(* Logix 5000 project; controller WWTP_SOLIDS_CLX vendor 1 type 14 code 54 rev 17.2; software revision 17.00; part 9 of 16 *)
(* tags used below, declared in another part *)
   Inp_RunFdbk : BOOL;   // Input Signal: RUN feedback from motor
   Inp_PermOK : BOOL;   // 1=Permissives OK, motor can start
   Inp_NBPermOK : BOOL;   // 1=Non-Bypassable Permissives OK, motor can start
   Inp_IntlkOK : BOOL;   // 1=Interlocks OK, motor can start/run
   Inp_NBIntlkOK : BOOL;   // 1=Non-Bypassable Interlocks OK, motor can start/run
   Inp_IOFault : BOOL;   // Input Communication Status 0=OK, 1=fail
   Inp_Sim : BOOL;   // 1=Simulate working motor; 0=Start/Stop/ Monitor actual motor
   Inp_Hand : BOOL;   // 1=Select Hand (hardwired) Control Strategy
   Inp_Ovrd : BOOL;   // 1=Select Override control strategy
   Inp_OvrdState : BOOL;   // 1=Override to RUN, 0=Override to STOP
   Inp_Reset : BOOL;   // 1=Reset all fault conditions and latched Alarms
   Cfg_HasRunFdbk : BOOL;   // 1=Motor provides a run feedback signal
   Cfg_UseRunFdbk : BOOL;   // 1=Motor run feedback should be used for failure checking
   Cfg_PCmdClear : BOOL;   // 1=Clear Program Commands on receipt 0=Leave Set
   Cfg_OvrdPermIntlk : BOOL;   // 1=Override ignores Bypassable Perm/ Intlk; 0=always use Perm/Intlk
   Cfg_HasFailToStartAlm : BOOL;   // 1=Fail to Start Alarm exists and will be checked
   Cfg_HasFailToStopAlm : BOOL;   // 1=Fail to Stop Alarm exists and will be checked
   Cfg_HasIntlkTripAlm : BOOL;   // 1=Interlock Trip Alarm exists and will be checked
   Cfg_HasIOFaultAlm : BOOL;   // 1=I/O Fault Alarm exists and will be checked
   Cfg_FailToStartResetReqd : BOOL;   // 1=Reset required to clear Fail to Start Alarm
   Cfg_FailToStopResetReqd : BOOL;   // 1=Reset required to clear Fail to Stop Alarm
   Cfg_IntlkTripResetReqd : BOOL;   // 1=Reset required to clear Interlock Trip Alarm
   Cfg_IOFaultResetReqd : BOOL;   // 1=Reset required to clear I/O Fault Alarm
   Cfg_FailToStartAckReqd : BOOL;   // 1=Acknowledge required for Fail to Start Alarm
   Cfg_FailToStopAckReqd : BOOL;   // 1=Acknowledge required for Fail to Stop Alarm
   Cfg_IntlkTripAckReqd : BOOL;   // 1=Acknowledge required for Interlock Trip Alarm
   Cfg_IOFaultAckReqd : BOOL;   // 1=Acknowledge required for I/O Fault Alarm
   Cfg_FailToStartSeverity : SINT;   // Fail To Start Alarm Severity 1=info 2=warn 3=excep 4=fault
   Cfg_FailToStopSeverity : SINT;   // Fail To Stop Alarm Severity 1=info 2=warn 3=excep 4=fault
   Cfg_IntlkTripSeverity : SINT;   // Interlock Trip Alarm Severity 1=info 2=warn 3=excep 4=fault
   Cfg_IOFaultSeverity : SINT;   // I/O Fault Alarm Severity 1=info 2=warn 3=excep 4=fault
   Cfg_SimFdbkT : DINT;   // Delay to echo back of Running/Stopped status when in Simulation (sec)
   Cfg_FailToStartT : DINT;   // Time after Start to get Run Feedback before Fault (sec)
   Cfg_FailToStopT : DINT;   // Time after Stop to drop Run Feedback before Fault (sec)
   PSet_Owner : DINT;   // Program Owner Request ID (non-zero) or Release (zero)
   PCmd_Start : BOOL;   // Program Command to Start Motor
   PCmd_Stop : BOOL;   // Program Command to Stop Motor
   PCmd_Acq : BOOL;   // Program Command to Acquire ownership (Oper/OOS to Prog)
   PCmd_Rel : BOOL;   // Program Command to Release ownership (Prog to OOS)
   PCmd_Lock : BOOL;   // Program Command to Lock Mode in Prog
   PCmd_Unlock : BOOL;   // Program Command to Unlock Mode
   PCmd_Reset : BOOL;   // Program Command to Reset all Alarms requiring Reset
   PCmd_FailToStartAck : BOOL;   // Program Command to Acknowledge Fail to Start Alarm
   PCmd_FailToStartInhibit : BOOL;   // Program Command to Inhibit Fail to Start Alarm
   PCmd_FailToStartUninhibit : BOOL;   // Program Command to Uninhibit Fail to Start Alarm
   PCmd_FailToStopAck : BOOL;   // Program Command to Acknowledge Fail to Stop Alarm
   PCmd_FailToStopInhibit : BOOL;   // Program Command to Inhibit Fail to Stop Alarm
   PCmd_FailToStopUninhibit : BOOL;   // Program Command to Uninhibit Fail to Stop Alarm
   PCmd_IntlkTripAck : BOOL;   // Program Command to Acknowledge Interlock Trip Alarm
   PCmd_IntlkTripInhibit : BOOL;   // Program Command to Inhibit Interlock Trip Alarm
   PCmd_IntlkTripUninhibit : BOOL;   // Program Command to Uninhibit Interlock Trip Alarm
   PCmd_IOFaultAck : BOOL;   // Program Command to Acknowledge I/O Fault Alarm
   PCmd_IOFaultInhibit : BOOL;   // Program Command to Inhibit I/O Fault Alarm
   PCmd_IOFaultUninhibit : BOOL;   // Program Command to Uninhibit I/O Fault Alarm
   OCmd_Start : BOOL;   // Operator Command to Start Motor
   OCmd_Stop : BOOL;   // Operator Command to Stop Motor
   OCmd_Bypass : BOOL;   // Operator Command to Bypass all Bypassable Interlocks and Permissives
   OCmd_Check : BOOL;   // Operator Command to Check (not bypass) all Interlocks and Permissives
   MCmd_Disable : BOOL;   // Maintenance Command to Disable Motor
   MCmd_Enable : BOOL;   // Maintenance Command to Enable (allow to run) Motor
   OCmd_Reset : BOOL;   // Operator Command to Reset all Alarms requiring Reset
   Out_Run : BOOL;   // 1=Run Motor, 0=Stop Motor
   Out_Start : BOOL;   // 1=Start Motor, 0=Motor left in current state
   Out_Stop : BOOL;   // 1=Stop Motor, 0=Motor left in current state
   Val_Owner : DINT;   // Current Object Owner ID (0=not owned)
   Val_Notify : SINT;   // Current Alarm Level and Acknowledgement (enumeration)
   Sts_Disabled : BOOL;   // 1=Motor is Disabled
   Sts_Err : BOOL;   // 1=Error in Config: see detail bits for reason
   Err_Timer : BOOL;   // 1=Error in Config: Start/Stop Check timer preset (use 0 to 2147483)
   Err_Sim : BOOL;   // 1=Error in Config: Simulation timer preset (use 0 to 2147483)
   Err_Alarm : BOOL;   // 1=Error in Config: Invalid Alarm Severity
   Sts_Hand : BOOL;   // 1=Mode is Hand (supersedes Maint, Ovrd, Prog, Oper)
   Sts_Maint : BOOL;   // 1=Mode is Maintenance (supersedes Ovrd, Prog, Oper)
   Sts_Ovrd : BOOL;   // 1=Mode is Override (supersedes Prog, Oper)
   Sts_Prog : BOOL;   // 1=Mode is Program (auto)
   Sts_Oper : BOOL;   // 1=Mode is Operator (manual)
   Sts_ProgOperLock : BOOL;   // 1=Program or Operator has requested Mode Lock
   Sts_FailToStart : BOOL;   // 1=Motor Failed to Start (one-shot)
   Alm_FailToStart : BOOL;   // 1=Motor Fail to Start Alarm
   Ack_FailToStart : BOOL;   // 1=Fail to Start Alarm has been acknowledged
   Sts_FailToStartDisabled : BOOL;   // 1=Fail to Start Alarm has been disabled (will not be sent)
   Sts_FailToStartInhibited : BOOL;   // 1=Fail to Start Alarm has been inhibited by logic
   Sts_FailToStartSuppressed : BOOL;   // 1=Fail to Start Alarm has been suppressed (logged only)
   Sts_FailToStop : BOOL;   // 1=Motor Failed to Stop
   Alm_FailToStop : BOOL;   // 1=Motor Fail to Stop Alarm
   Ack_FailToStop : BOOL;   // 1=Fail to Stop Alarm has been acknowledged
   Sts_FailToStopDisabled : BOOL;   // 1=Fail to Stop Alarm has been disabled (will not be sent)
   Sts_FailToStopInhibited : BOOL;   // 1=Fail to Stop Alarm has been inhibited by logic
   Sts_FailToStopSuppressed : BOOL;   // 1=Fail to Stop Alarm has been suppressed (logged only)
   Sts_IntlkTrip : BOOL;   // 1=Motor stopped by an Interlock NOT OK (one-shot)
   Sts_IOFault : BOOL;   // I/O Comm Fault Status (0=OK, 1=Bad)
   Rdy_Reset : BOOL;   // 1=Ready to receive OCmd_Reset (enables HMI button)
   Mode : P_Mode;   // Motor Mode Selection
   IOFault : P_Alarm;   // I/O Fault Alarm
   IntlkTrip : P_Alarm;   // Interlock Trip Alarm
   FailToStop : P_Alarm;   // Motor Failed to Stop Alarm
   FailToStart : P_Alarm;   // Motor Failed to Start Alarm
   Wrk_Run : BOOL;   // 1=Motor should be "running", 0=should be "stopped"
   Wrk_SimRunT : TIMER;   // Simulation Delay until Running
   Wrk_StopT : TIMER;   // Stop Check Timer
   Wrk_StartT : TIMER;   // Start Check Timer
   Wrk_Fault : BOOL;   // 1=a Motor Fault has been detected
   Wrk_SimStopT : TIMER;   // Simulation Delay until Stopped
   Wrk_RunFdbk : BOOL;   // Run Feedback based on mode, simulation, etc. 1=running
   Wrk_IntlkTrip : BOOL;   // 1=Interlock Not OK Tripped Running Motor
   Wrk_Bypass : BOOL;   // Internal Bypassable Permissives and Interlocks are Bypassed flag
   Wrk_Disabled : BOOL;   // Internal Motor is Disabled
(* P_Motor, continued *)

ROUTINE Logic   (* ladder *)
// Normal Scan: control / monitor single speed motor
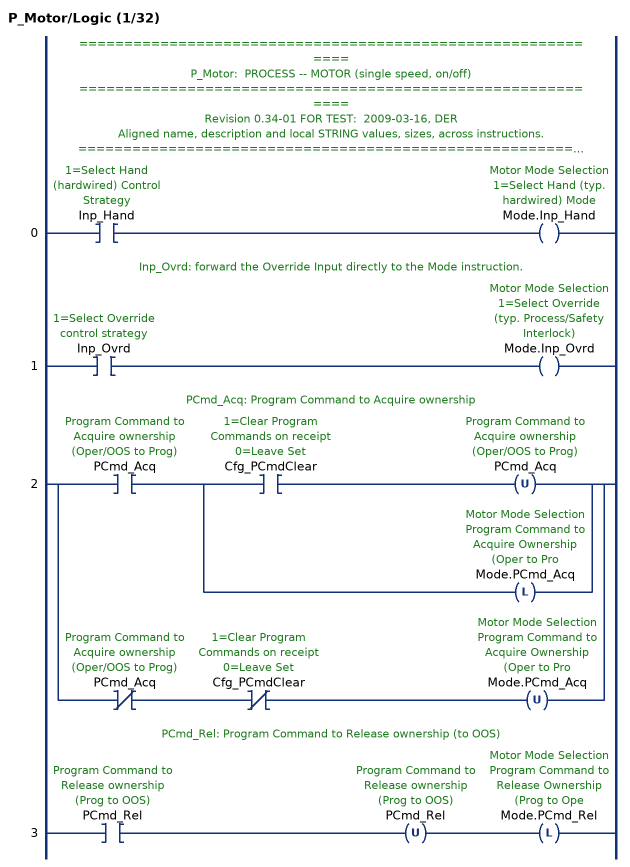
   // ============================================================
   // P_Motor:  PROCESS -- MOTOR (single speed, on/off)
   // ============================================================
   // Revision 0.34-01 FOR TEST:  2009-03-16, DER
   // Aligned name, description and local STRING values, sizes, across instructions.
   // ============================================================
   // This Instruction controls and monitors a single-speed motor
   // (FVNR, soft-start, etc.) and provides:
   // *  Monitoring of run feedback, display of actual motor status
   // *  Detection of Failure to Start, Failure to Stop
   // *  Monitoring of a Permissive condition to allow starting
   // * Monitoring of an Interlock condition to stop / prevent starting
   // * Simulation, providing feedback of a working motor while disabling outputs
   // * Monitoring of I/O communication faults
   // * Alarms for Fail to Start, Fail to Stop, Interlock Trip, I/O Fault
   // * Operation in Hand, Maintenance, Override, Program and Operator Modes
   // * "Available" status for use by automation logic to know whether motor
   // can be controlled by other objects.
   // ============================================================
   // POWERUP / INVALID STATE HANDLING
   // ============================================================
   // Mode states are retained through a power cycle.
   // Motor "run" request is cleared on first scan, in the rung which unlatches "Wrk_Run", below
   // ============================================================
   // MODE PROCESSING
   // ============================================================
   // These rungs handle received Mode Inputs and Commands:
   // NOTE:  Operator Commands for Mode, Alarm are sent directly to the contained P_Mode and P_Alarm AOIs.
   // Inp_Hand: forward the Hand Input directly to the Mode instruction.
   0: XIC(Inp_Hand)OTE(Mode.Inp_Hand);
   // Inp_Ovrd: forward the Override Input directly to the Mode instruction.
   1: XIC(Inp_Ovrd)OTE(Mode.Inp_Ovrd);
   // PCmd_Acq: Program Command to Acquire ownership
   2: [XIC(PCmd_Acq) [XIC(Cfg_PCmdClear) OTU(PCmd_Acq) ,OTL(Mode.PCmd_Acq) ] ,XIO(PCmd_Acq) XIO(Cfg_PCmdClear) OTU(Mode.PCmd_Acq) ];
   // PCmd_Rel: Program Command to Release ownership (to OOS)
   3: XIC(PCmd_Rel)OTU(PCmd_Rel)OTL(Mode.PCmd_Rel);
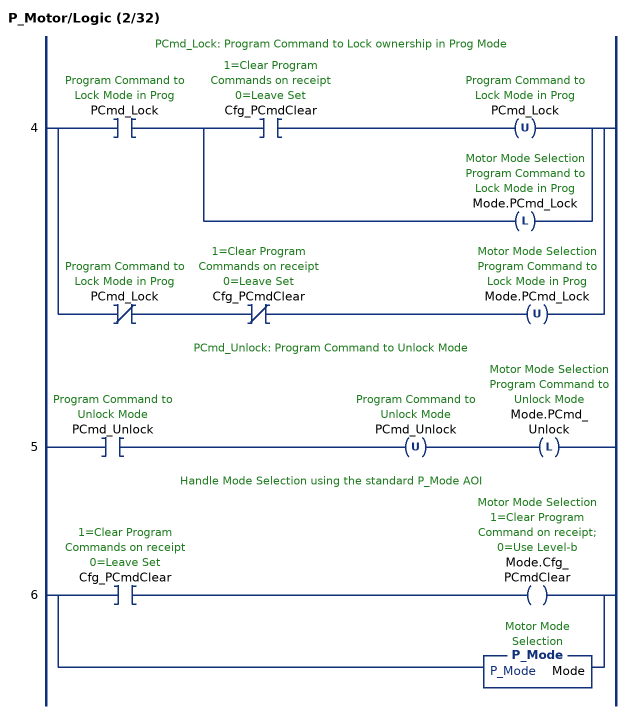
   // PCmd_Lock: Program Command to Lock ownership in Prog Mode
   4: [XIC(PCmd_Lock) [XIC(Cfg_PCmdClear) OTU(PCmd_Lock) ,OTL(Mode.PCmd_Lock) ] ,XIO(PCmd_Lock) XIO(Cfg_PCmdClear) OTU(Mode.PCmd_Lock) ];
   // PCmd_Unlock: Program Command to Unlock Mode
   5: XIC(PCmd_Unlock)OTU(PCmd_Unlock)OTL(Mode.PCmd_Unlock);
   // Handle Mode Selection using the standard P_Mode AOI
   6: [XIC(Cfg_PCmdClear) OTE(Mode.Cfg_PCmdClear) ,P_Mode(Mode) ];
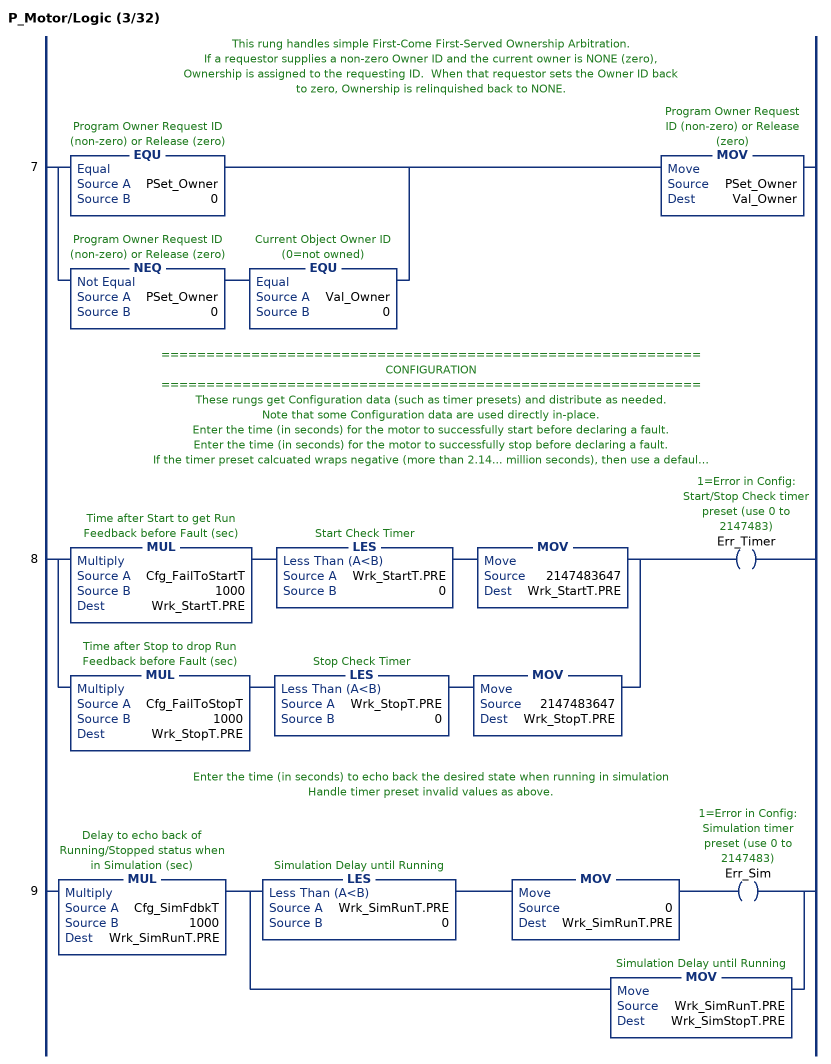
   // This rung handles simple First-Come First-Served Ownership Arbitration.
   // If a requestor supplies a non-zero Owner ID and the current owner is NONE (zero),
   // Ownership is assigned to the requesting ID.  When that requestor sets the Owner ID back
   // to zero, Ownership is relinquished back to NONE.
   7: [EQU(PSet_Owner,0) ,NEQ(PSet_Owner,0) EQU(Val_Owner,0) ]MOV(PSet_Owner,Val_Owner);
   // ============================================================
   // CONFIGURATION
   // ============================================================
   // These rungs get Configuration data (such as timer presets) and distribute as needed.
   // Note that some Configuration data are used directly in-place.
   // Enter the time (in seconds) for the motor to successfully start before declaring a fault.
   // Enter the time (in seconds) for the motor to successfully stop before declaring a fault.
   // If the timer preset calcuated wraps negative (more than 2.14... million seconds), then use a default
   // limit value and report Bad Configuration.  Note that a negative timer preset will fault the controller!!!
   8: [MUL(Cfg_FailToStartT,1000,Wrk_StartT.PRE) LES(Wrk_StartT.PRE,0) MOV(2147483647,Wrk_StartT.PRE) ,MUL(Cfg_FailToStopT,1000,Wrk_StopT.PRE) LES(Wrk_StopT.PRE,0) MOV(2147483647,Wrk_StopT.PRE) ]OTE(Err_Timer);
   // Enter the time (in seconds) to echo back the desired state when running in simulation
   // Handle timer preset invalid values as above.
   9: MUL(Cfg_SimFdbkT,1000,Wrk_SimRunT.PRE)[LES(Wrk_SimRunT.PRE,0) MOV(0,Wrk_SimRunT.PRE) OTE(Err_Sim) ,MOV(Wrk_SimRunT.PRE,Wrk_SimStopT.PRE) ];
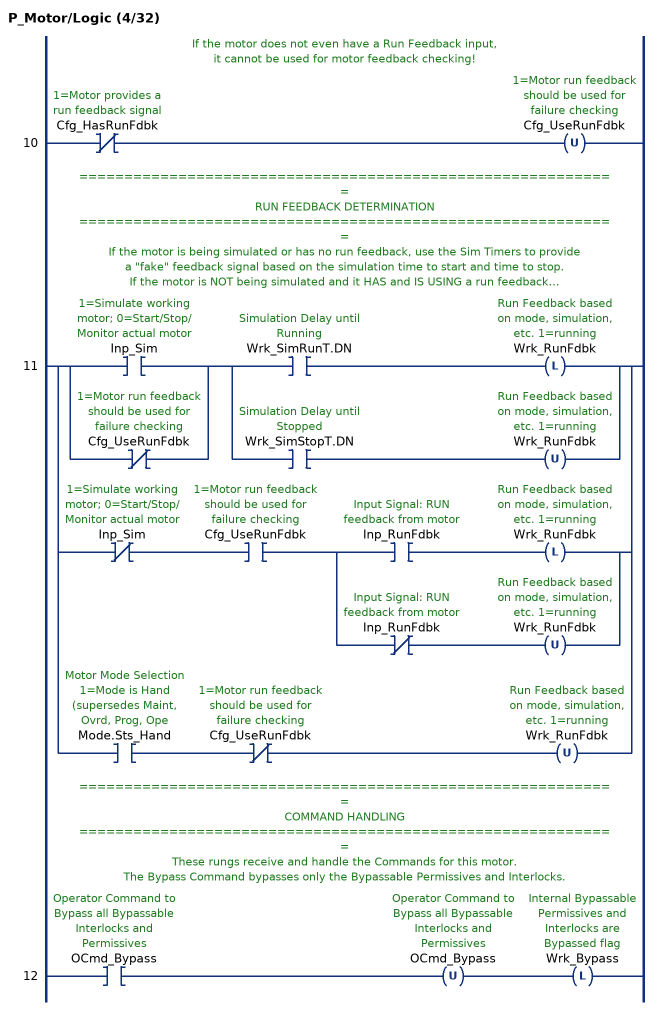
   // If the motor does not even have a Run Feedback input,
   // it cannot be used for motor feedback checking!
   10: XIO(Cfg_HasRunFdbk)OTU(Cfg_UseRunFdbk);
   // ============================================================
   // RUN FEEDBACK DETERMINATION
   // ============================================================
   // If the motor is being simulated or has no run feedback, use the Sim Timers to provide
   // a "fake" feedback signal based on the simulation time to start and time to stop.
   // If the motor is NOT being simulated and it HAS and IS USING a run feedback,
   // use the state of the run feedback input as the motor run state.
   11: [[XIC(Inp_Sim) ,XIO(Cfg_UseRunFdbk) ] [XIC(Wrk_SimRunT.DN) OTL(Wrk_RunFdbk) ,XIC(Wrk_SimStopT.DN) OTU(Wrk_RunFdbk) ] ,XIO(Inp_Sim) XIC(Cfg_UseRunFdbk) [XIC(Inp_RunFdbk) OTL(Wrk_RunFdbk) ,XIO(Inp_RunFdbk) OTU(Wrk_RunFdbk) ] ,XIC(Mode.Sts_Hand) XIO(Cfg_UseRunFdbk) OTU(Wrk_RunFdbk) ];
   // ============================================================
   // COMMAND HANDLING
   // ============================================================
   // These rungs receive and handle the Commands for this motor.
   // The Bypass Command bypasses only the Bypassable Permissives and Interlocks.
   12: XIC(OCmd_Bypass)OTU(OCmd_Bypass)OTL(Wrk_Bypass);
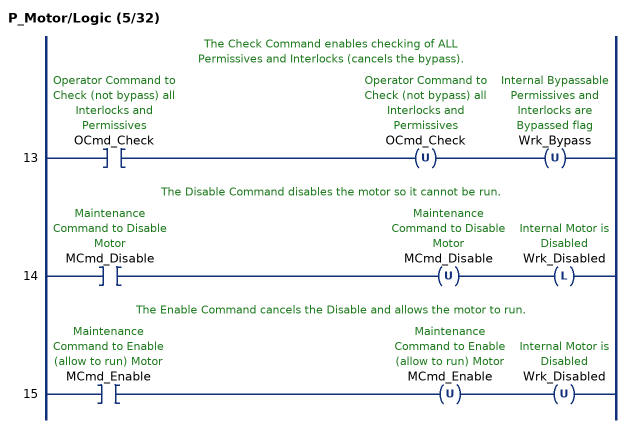
   // The Check Command enables checking of ALL
   // Permissives and Interlocks (cancels the bypass).
   13: XIC(OCmd_Check)OTU(OCmd_Check)OTU(Wrk_Bypass);
   // The Disable Command disables the motor so it cannot be run.
   14: XIC(MCmd_Disable)OTU(MCmd_Disable)OTL(Wrk_Disabled);
   // The Enable Command cancels the Disable and allows the motor to run.
   15: XIC(MCmd_Enable)OTU(MCmd_Enable)OTU(Wrk_Disabled);
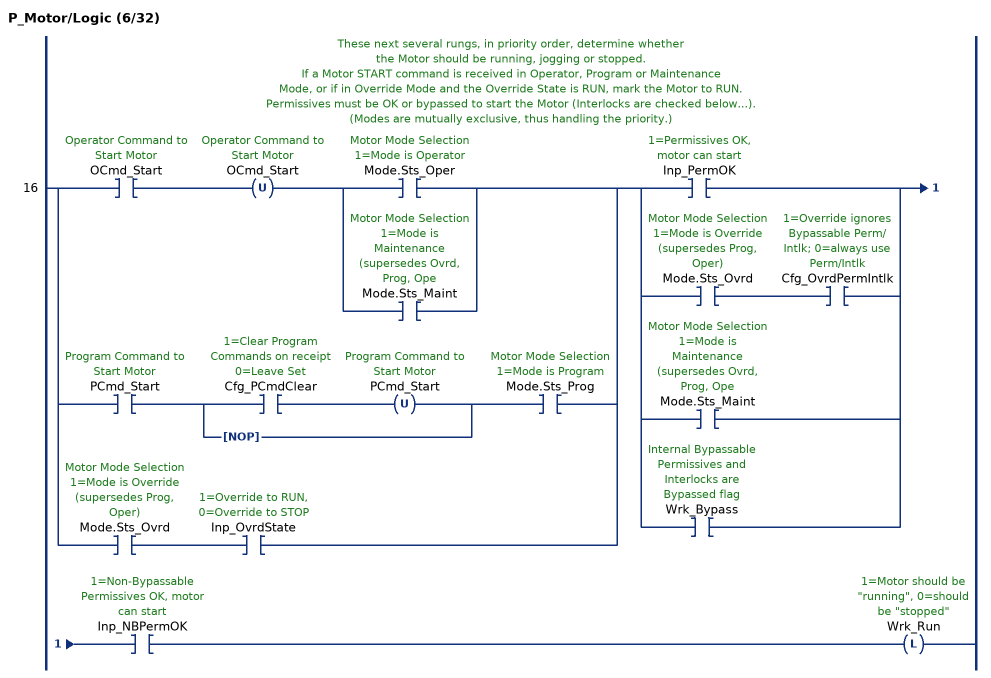
   // These next several rungs, in priority order, determine whether
   // the Motor should be running, jogging or stopped.
   // If a Motor START command is received in Operator, Program or Maintenance
   // Mode, or if in Override Mode and the Override State is RUN, mark the Motor to RUN.
   // Permissives must be OK or bypassed to start the Motor (Interlocks are checked below...).
   // (Modes are mutually exclusive, thus handling the priority.)
   16: [XIC(OCmd_Start) OTU(OCmd_Start) [XIC(Mode.Sts_Oper) ,XIC(Mode.Sts_Maint) ] ,XIC(PCmd_Start) [XIC(Cfg_PCmdClear) OTU(PCmd_Start) ,NOP() ] XIC(Mode.Sts_Prog) ,XIC(Mode.Sts_Ovrd) XIC(Inp_OvrdState) ][XIC(Inp_PermOK) ,XIC(Mode.Sts_Ovrd) XIC(Cfg_OvrdPermIntlk) ,XIC(Mode.Sts_Maint) ,XIC(Wrk_Bypass) ]XIC(Inp_NBPermOK)OTL(Wrk_Run);
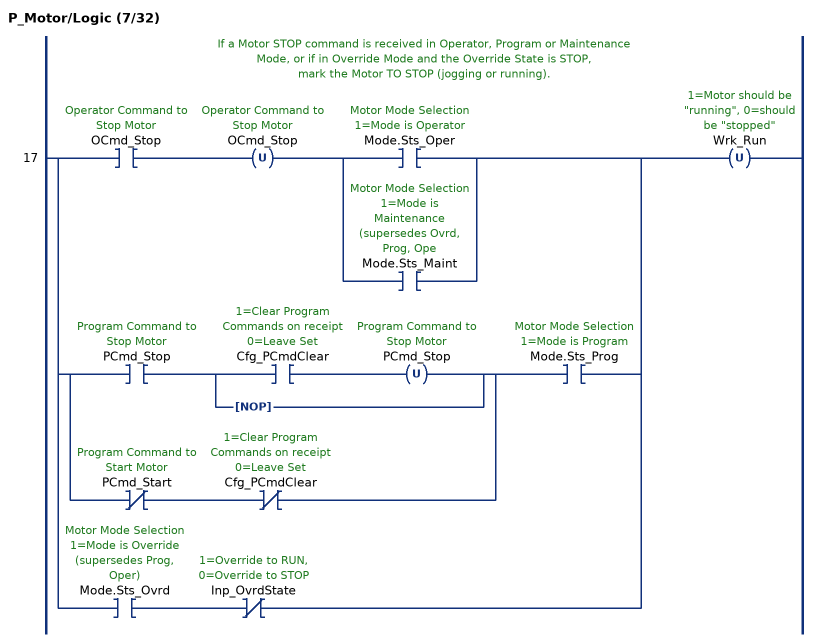
   // If a Motor STOP command is received in Operator, Program or Maintenance
   // Mode, or if in Override Mode and the Override State is STOP,
   // mark the Motor TO STOP (jogging or running).
   17: [XIC(OCmd_Stop) OTU(OCmd_Stop) [XIC(Mode.Sts_Oper) ,XIC(Mode.Sts_Maint) ] ,[XIC(PCmd_Stop) [XIC(Cfg_PCmdClear) OTU(PCmd_Stop) ,NOP() ] ,XIO(PCmd_Start) XIO(Cfg_PCmdClear) ] XIC(Mode.Sts_Prog) ,XIC(Mode.Sts_Ovrd) XIO(Inp_OvrdState) ]OTU(Wrk_Run);
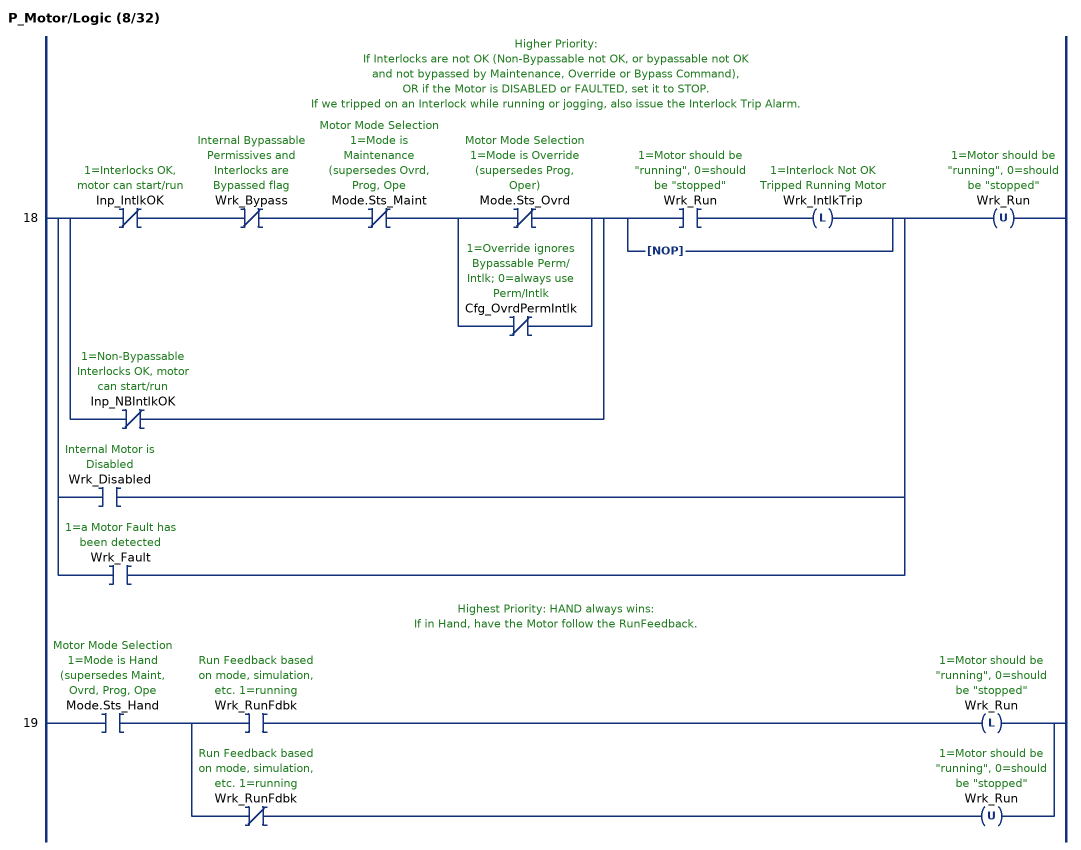
   // Higher Priority:
   // If Interlocks are not OK (Non-Bypassable not OK, or bypassable not OK
   // and not bypassed by Maintenance, Override or Bypass Command),
   // OR if the Motor is DISABLED or FAULTED, set it to STOP.
   // If we tripped on an Interlock while running or jogging, also issue the Interlock Trip Alarm.
   18: [[XIO(Inp_IntlkOK) XIO(Wrk_Bypass) XIO(Mode.Sts_Maint) [XIO(Mode.Sts_Ovrd) ,XIO(Cfg_OvrdPermIntlk) ] ,XIO(Inp_NBIntlkOK) ] [XIC(Wrk_Run) OTL(Wrk_IntlkTrip) ,NOP() ] ,XIC(Wrk_Disabled) ,XIC(Wrk_Fault) ]OTU(Wrk_Run);
   // Highest Priority: HAND always wins:
   // If in Hand, have the Motor follow the RunFeedback.
   19: XIC(Mode.Sts_Hand)[XIC(Wrk_RunFdbk) OTL(Wrk_Run) ,XIO(Wrk_RunFdbk) OTU(Wrk_Run) ];
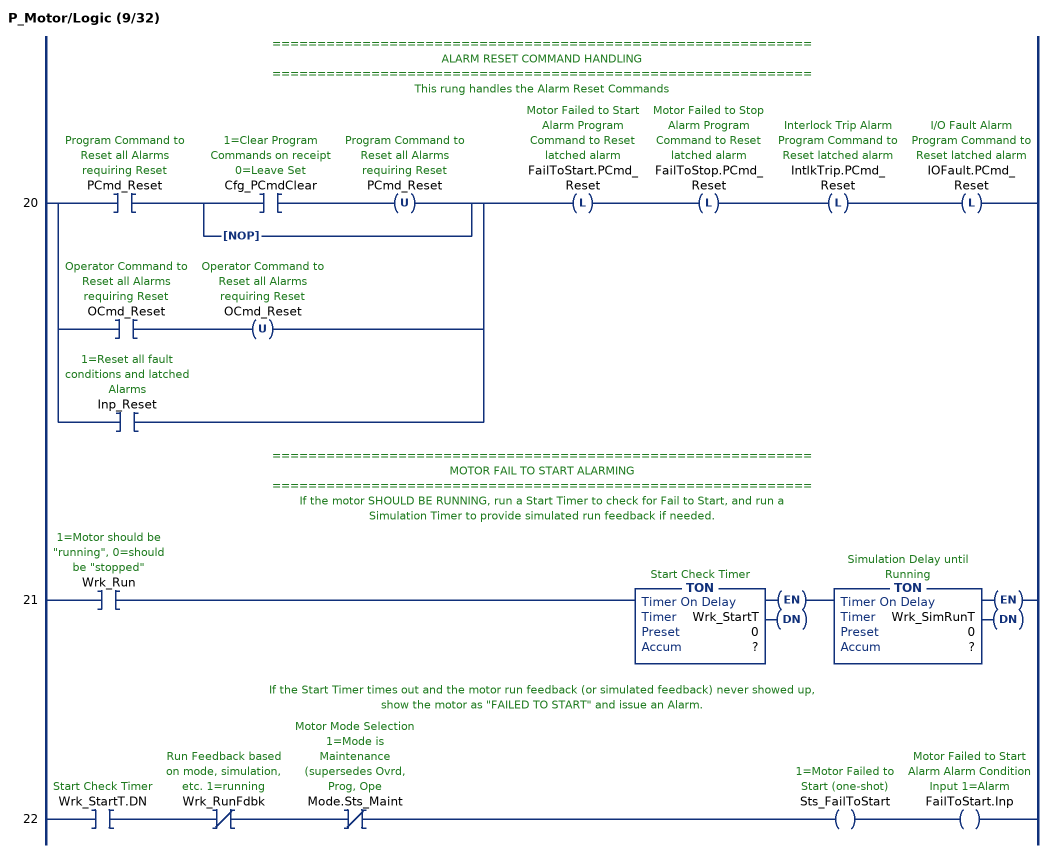
   // ============================================================
   // ALARM RESET COMMAND HANDLING
   // ============================================================
   // This rung handles the Alarm Reset Commands
   20: [XIC(PCmd_Reset) [XIC(Cfg_PCmdClear) OTU(PCmd_Reset) ,NOP() ] ,XIC(OCmd_Reset) OTU(OCmd_Reset) ,XIC(Inp_Reset) ]OTL(FailToStart.PCmd_Reset)OTL(FailToStop.PCmd_Reset)OTL(IntlkTrip.PCmd_Reset)OTL(IOFault.PCmd_Reset);
   // ============================================================
   // MOTOR FAIL TO START ALARMING
   // ============================================================
   // If the motor SHOULD BE RUNNING, run a Start Timer to check for Fail to Start, and run a
   // Simulation Timer to provide simulated run feedback if needed.
   21: XIC(Wrk_Run)TON(Wrk_StartT,?,?)TON(Wrk_SimRunT,?,?);
   // If the Start Timer times out and the motor run feedback (or simulated feedback) never showed up,
   // show the motor as "FAILED TO START" and issue an Alarm.
   22: XIC(Wrk_StartT.DN)XIO(Wrk_RunFdbk)XIO(Mode.Sts_Maint)OTE(Sts_FailToStart)OTE(FailToStart.Inp);
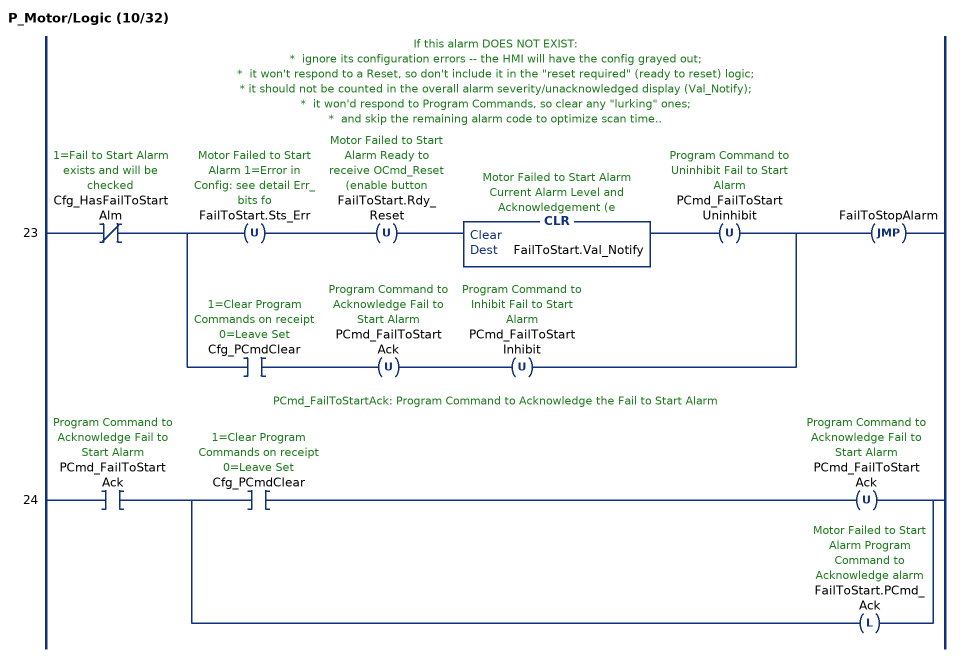
   // If this alarm DOES NOT EXIST:
   // *  ignore its configuration errors -- the HMI will have the config grayed out;
   // *  it won't respond to a Reset, so don't include it in the "reset required" (ready to reset) logic;
   // * it should not be counted in the overall alarm severity/unacknowledged display (Val_Notify);
   // *  it won'd respond to Program Commands, so clear any "lurking" ones;
   // *  and skip the remaining alarm code to optimize scan time..
   23: XIO(Cfg_HasFailToStartAlm)[OTU(FailToStart.Sts_Err) OTU(FailToStart.Rdy_Reset) CLR(FailToStart.Val_Notify) OTU(PCmd_FailToStartUninhibit) ,XIC(Cfg_PCmdClear) OTU(PCmd_FailToStartAck) OTU(PCmd_FailToStartInhibit) ]JMP(FailToStopAlarm);
   // PCmd_FailToStartAck: Program Command to Acknowledge the Fail to Start Alarm
   24: XIC(PCmd_FailToStartAck)[XIC(Cfg_PCmdClear) OTU(PCmd_FailToStartAck) ,OTL(FailToStart.PCmd_Ack) ];
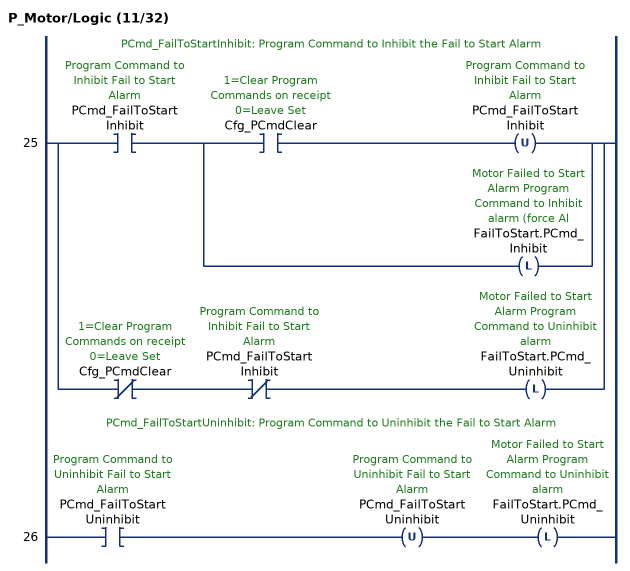
   // PCmd_FailToStartInhibit: Program Command to Inhibit the Fail to Start Alarm
   25: [XIC(PCmd_FailToStartInhibit) [XIC(Cfg_PCmdClear) OTU(PCmd_FailToStartInhibit) ,OTL(FailToStart.PCmd_Inhibit) ] ,XIO(Cfg_PCmdClear) XIO(PCmd_FailToStartInhibit) OTL(FailToStart.PCmd_Uninhibit) ];
   // PCmd_FailToStartUninhibit: Program Command to Uninhibit the Fail to Start Alarm
   26: XIC(PCmd_FailToStartUninhibit)OTU(PCmd_FailToStartUninhibit)OTL(FailToStart.PCmd_Uninhibit);
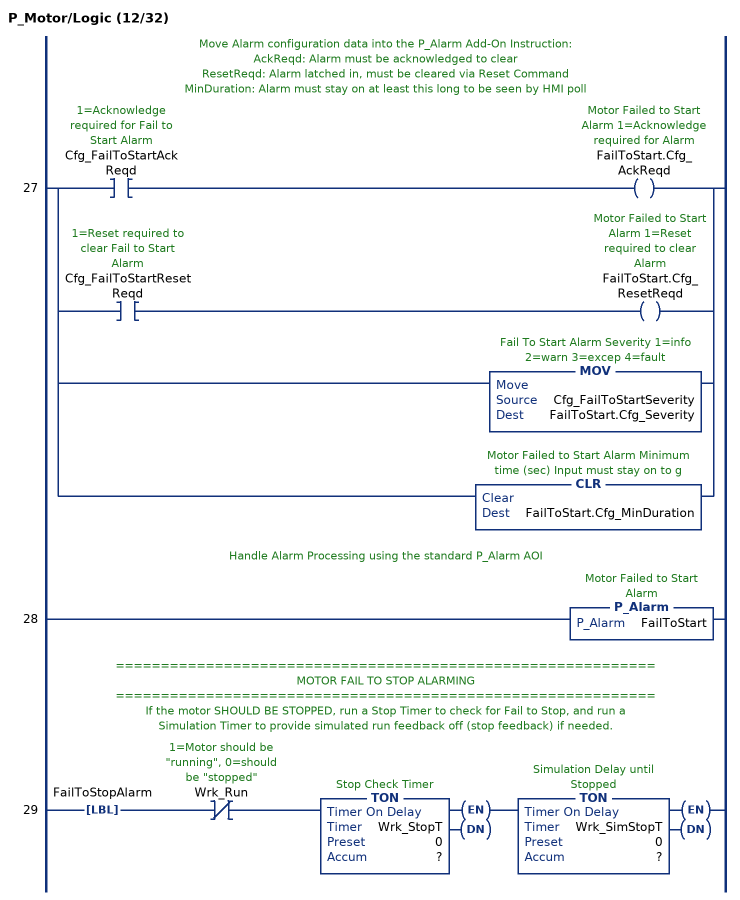
   // Move Alarm configuration data into the P_Alarm Add-On Instruction:
   // AckReqd: Alarm must be acknowledged to clear
   // ResetReqd: Alarm latched in, must be cleared via Reset Command
   // MinDuration: Alarm must stay on at least this long to be seen by HMI poll
   27: [XIC(Cfg_FailToStartAckReqd) OTE(FailToStart.Cfg_AckReqd) ,XIC(Cfg_FailToStartResetReqd) OTE(FailToStart.Cfg_ResetReqd) ,MOV(Cfg_FailToStartSeverity,FailToStart.Cfg_Severity) ,CLR(FailToStart.Cfg_MinDuration) ];
   // Handle Alarm Processing using the standard P_Alarm AOI
   28: P_Alarm(FailToStart);
   // ============================================================
   // MOTOR FAIL TO STOP ALARMING
   // ============================================================
   // If the motor SHOULD BE STOPPED, run a Stop Timer to check for Fail to Stop, and run a
   // Simulation Timer to provide simulated run feedback off (stop feedback) if needed.
   29: LBL(FailToStopAlarm)XIO(Wrk_Run)TON(Wrk_StopT,?,?)TON(Wrk_SimStopT,?,?);
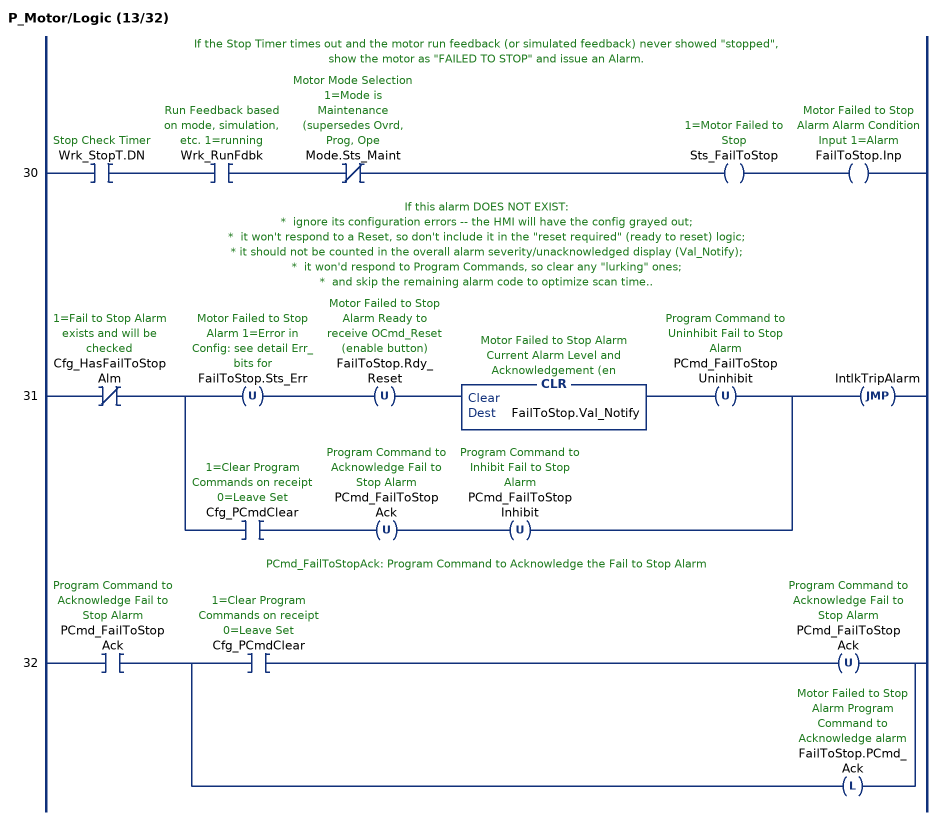
   // If the Stop Timer times out and the motor run feedback (or simulated feedback) never showed "stopped",
   // show the motor as "FAILED TO STOP" and issue an Alarm.
   30: XIC(Wrk_StopT.DN)XIC(Wrk_RunFdbk)XIO(Mode.Sts_Maint)OTE(Sts_FailToStop)OTE(FailToStop.Inp);
   // If this alarm DOES NOT EXIST:
   // *  ignore its configuration errors -- the HMI will have the config grayed out;
   // *  it won't respond to a Reset, so don't include it in the "reset required" (ready to reset) logic;
   // * it should not be counted in the overall alarm severity/unacknowledged display (Val_Notify);
   // *  it won'd respond to Program Commands, so clear any "lurking" ones;
   // *  and skip the remaining alarm code to optimize scan time..
   31: XIO(Cfg_HasFailToStopAlm)[OTU(FailToStop.Sts_Err) OTU(FailToStop.Rdy_Reset) CLR(FailToStop.Val_Notify) OTU(PCmd_FailToStopUninhibit) ,XIC(Cfg_PCmdClear) OTU(PCmd_FailToStopAck) OTU(PCmd_FailToStopInhibit) ]JMP(IntlkTripAlarm);
   // PCmd_FailToStopAck: Program Command to Acknowledge the Fail to Stop Alarm
   32: XIC(PCmd_FailToStopAck)[XIC(Cfg_PCmdClear) OTU(PCmd_FailToStopAck) ,OTL(FailToStop.PCmd_Ack) ];
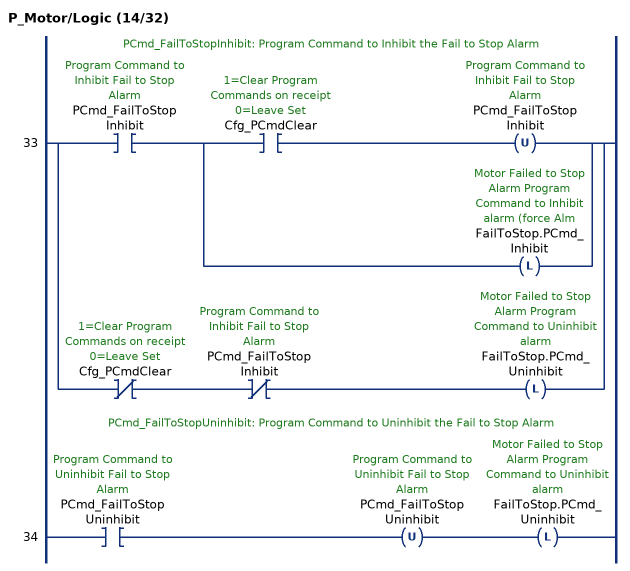
   // PCmd_FailToStopInhibit: Program Command to Inhibit the Fail to Stop Alarm
   33: [XIC(PCmd_FailToStopInhibit) [XIC(Cfg_PCmdClear) OTU(PCmd_FailToStopInhibit) ,OTL(FailToStop.PCmd_Inhibit) ] ,XIO(Cfg_PCmdClear) XIO(PCmd_FailToStopInhibit) OTL(FailToStop.PCmd_Uninhibit) ];
   // PCmd_FailToStopUninhibit: Program Command to Uninhibit the Fail to Stop Alarm
   34: XIC(PCmd_FailToStopUninhibit)OTU(PCmd_FailToStopUninhibit)OTL(FailToStop.PCmd_Uninhibit);
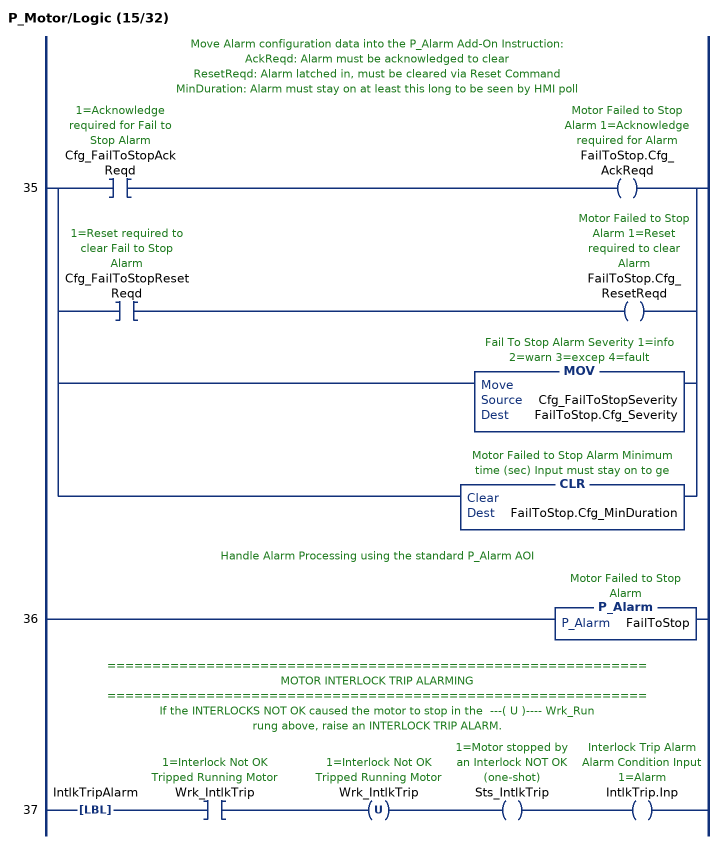
   // Move Alarm configuration data into the P_Alarm Add-On Instruction:
   // AckReqd: Alarm must be acknowledged to clear
   // ResetReqd: Alarm latched in, must be cleared via Reset Command
   // MinDuration: Alarm must stay on at least this long to be seen by HMI poll
   35: [XIC(Cfg_FailToStopAckReqd) OTE(FailToStop.Cfg_AckReqd) ,XIC(Cfg_FailToStopResetReqd) OTE(FailToStop.Cfg_ResetReqd) ,MOV(Cfg_FailToStopSeverity,FailToStop.Cfg_Severity) ,CLR(FailToStop.Cfg_MinDuration) ];
   // Handle Alarm Processing using the standard P_Alarm AOI
   36: P_Alarm(FailToStop);
   // ============================================================
   // MOTOR INTERLOCK TRIP ALARMING
   // ============================================================
   // If the INTERLOCKS NOT OK caused the motor to stop in the  ---( U )---- Wrk_Run
   // rung above, raise an INTERLOCK TRIP ALARM.
   37: LBL(IntlkTripAlarm)XIC(Wrk_IntlkTrip)OTU(Wrk_IntlkTrip)OTE(Sts_IntlkTrip)OTE(IntlkTrip.Inp);
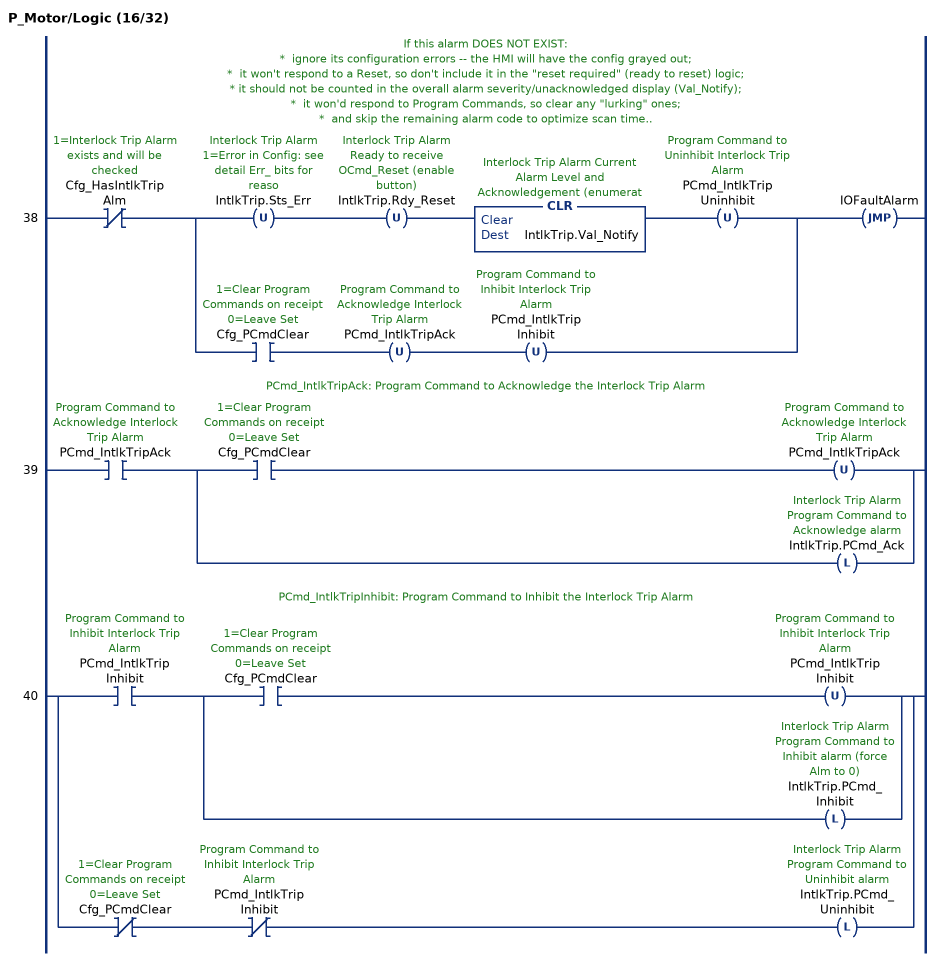
   // If this alarm DOES NOT EXIST:
   // *  ignore its configuration errors -- the HMI will have the config grayed out;
   // *  it won't respond to a Reset, so don't include it in the "reset required" (ready to reset) logic;
   // * it should not be counted in the overall alarm severity/unacknowledged display (Val_Notify);
   // *  it won'd respond to Program Commands, so clear any "lurking" ones;
   // *  and skip the remaining alarm code to optimize scan time..
   38: XIO(Cfg_HasIntlkTripAlm)[OTU(IntlkTrip.Sts_Err) OTU(IntlkTrip.Rdy_Reset) CLR(IntlkTrip.Val_Notify) OTU(PCmd_IntlkTripUninhibit) ,XIC(Cfg_PCmdClear) OTU(PCmd_IntlkTripAck) OTU(PCmd_IntlkTripInhibit) ]JMP(IOFaultAlarm);
   // PCmd_IntlkTripAck: Program Command to Acknowledge the Interlock Trip Alarm
   39: XIC(PCmd_IntlkTripAck)[XIC(Cfg_PCmdClear) OTU(PCmd_IntlkTripAck) ,OTL(IntlkTrip.PCmd_Ack) ];
   // PCmd_IntlkTripInhibit: Program Command to Inhibit the Interlock Trip Alarm
   40: [XIC(PCmd_IntlkTripInhibit) [XIC(Cfg_PCmdClear) OTU(PCmd_IntlkTripInhibit) ,OTL(IntlkTrip.PCmd_Inhibit) ] ,XIO(Cfg_PCmdClear) XIO(PCmd_IntlkTripInhibit) OTL(IntlkTrip.PCmd_Uninhibit) ];
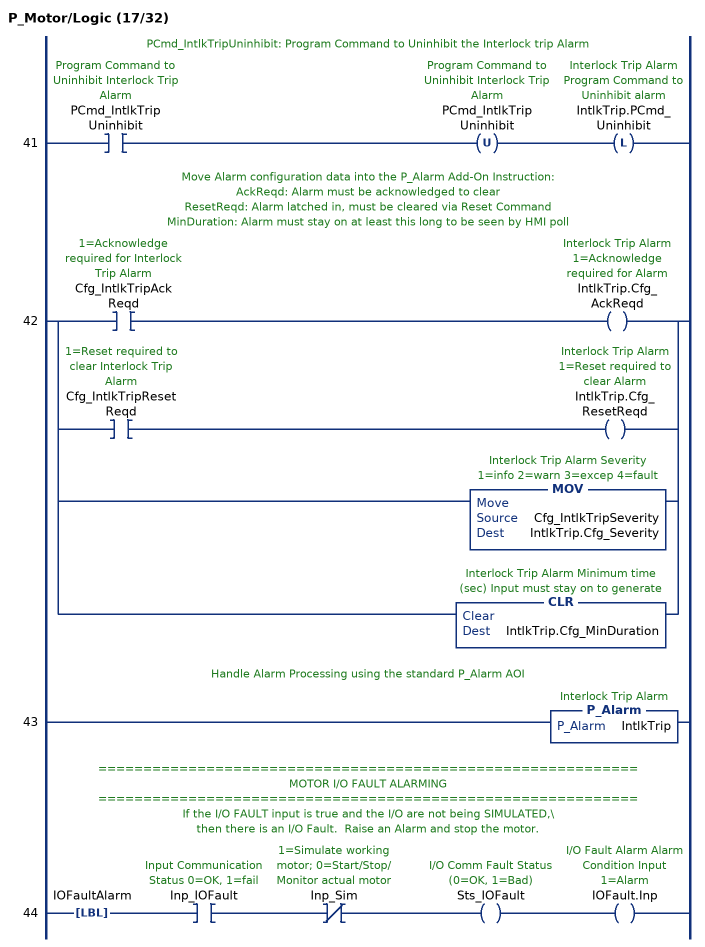
   // PCmd_IntlkTripUninhibit: Program Command to Uninhibit the Interlock trip Alarm
   41: XIC(PCmd_IntlkTripUninhibit)OTU(PCmd_IntlkTripUninhibit)OTL(IntlkTrip.PCmd_Uninhibit);
   // Move Alarm configuration data into the P_Alarm Add-On Instruction:
   // AckReqd: Alarm must be acknowledged to clear
   // ResetReqd: Alarm latched in, must be cleared via Reset Command
   // MinDuration: Alarm must stay on at least this long to be seen by HMI poll
   42: [XIC(Cfg_IntlkTripAckReqd) OTE(IntlkTrip.Cfg_AckReqd) ,XIC(Cfg_IntlkTripResetReqd) OTE(IntlkTrip.Cfg_ResetReqd) ,MOV(Cfg_IntlkTripSeverity,IntlkTrip.Cfg_Severity) ,CLR(IntlkTrip.Cfg_MinDuration) ];
   // Handle Alarm Processing using the standard P_Alarm AOI
   43: P_Alarm(IntlkTrip);
   // ============================================================
   // MOTOR I/O FAULT ALARMING
   // ============================================================
   // If the I/O FAULT input is true and the I/O are not being SIMULATED,\
   // then there is an I/O Fault.  Raise an Alarm and stop the motor.
   44: LBL(IOFaultAlarm)XIC(Inp_IOFault)XIO(Inp_Sim)OTE(Sts_IOFault)OTE(IOFault.Inp);
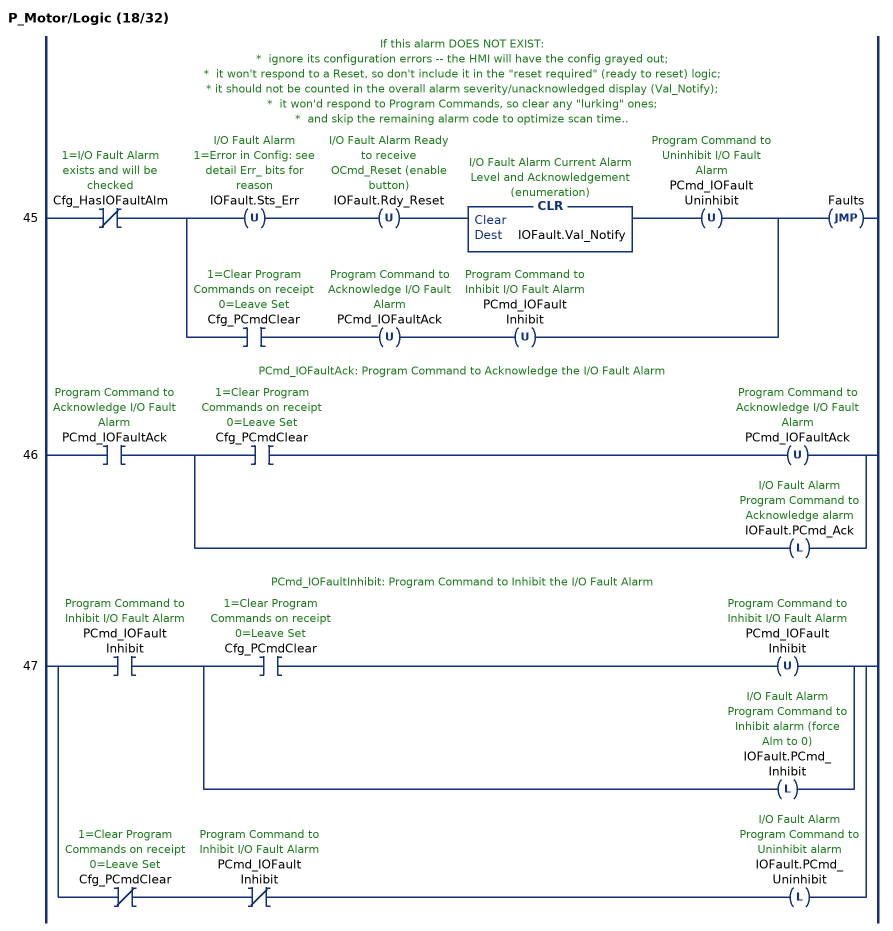
   // If this alarm DOES NOT EXIST:
   // *  ignore its configuration errors -- the HMI will have the config grayed out;
   // *  it won't respond to a Reset, so don't include it in the "reset required" (ready to reset) logic;
   // * it should not be counted in the overall alarm severity/unacknowledged display (Val_Notify);
   // *  it won'd respond to Program Commands, so clear any "lurking" ones;
   // *  and skip the remaining alarm code to optimize scan time..
   45: XIO(Cfg_HasIOFaultAlm)[OTU(IOFault.Sts_Err) OTU(IOFault.Rdy_Reset) CLR(IOFault.Val_Notify) OTU(PCmd_IOFaultUninhibit) ,XIC(Cfg_PCmdClear) OTU(PCmd_IOFaultAck) OTU(PCmd_IOFaultInhibit) ]JMP(Faults);
   // PCmd_IOFaultAck: Program Command to Acknowledge the I/O Fault Alarm
   46: XIC(PCmd_IOFaultAck)[XIC(Cfg_PCmdClear) OTU(PCmd_IOFaultAck) ,OTL(IOFault.PCmd_Ack) ];
   // PCmd_IOFaultInhibit: Program Command to Inhibit the I/O Fault Alarm
   47: [XIC(PCmd_IOFaultInhibit) [XIC(Cfg_PCmdClear) OTU(PCmd_IOFaultInhibit) ,OTL(IOFault.PCmd_Inhibit) ] ,XIO(Cfg_PCmdClear) XIO(PCmd_IOFaultInhibit) OTL(IOFault.PCmd_Uninhibit) ];
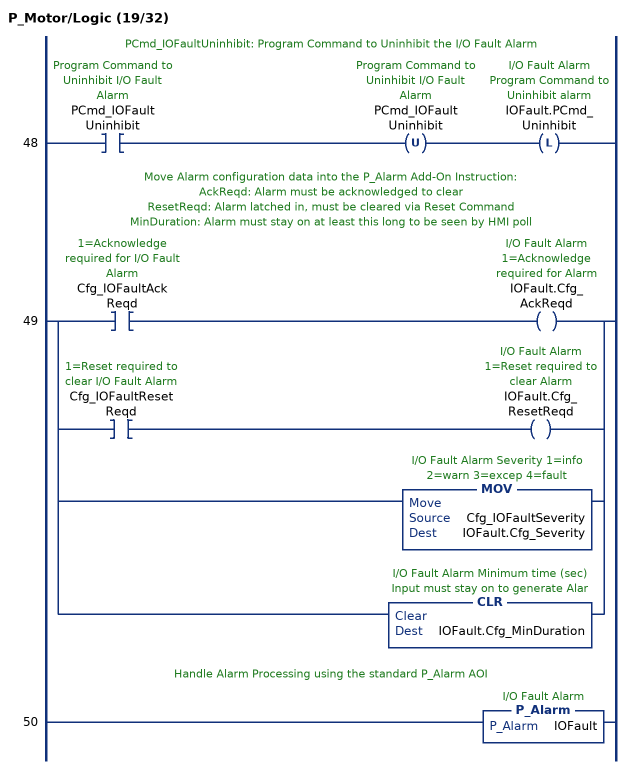
   // PCmd_IOFaultUninhibit: Program Command to Uninhibit the I/O Fault Alarm
   48: XIC(PCmd_IOFaultUninhibit)OTU(PCmd_IOFaultUninhibit)OTL(IOFault.PCmd_Uninhibit);
   // Move Alarm configuration data into the P_Alarm Add-On Instruction:
   // AckReqd: Alarm must be acknowledged to clear
   // ResetReqd: Alarm latched in, must be cleared via Reset Command
   // MinDuration: Alarm must stay on at least this long to be seen by HMI poll
   49: [XIC(Cfg_IOFaultAckReqd) OTE(IOFault.Cfg_AckReqd) ,XIC(Cfg_IOFaultResetReqd) OTE(IOFault.Cfg_ResetReqd) ,MOV(Cfg_IOFaultSeverity,IOFault.Cfg_Severity) ,CLR(IOFault.Cfg_MinDuration) ];
   // Handle Alarm Processing using the standard P_Alarm AOI
   50: P_Alarm(IOFault);
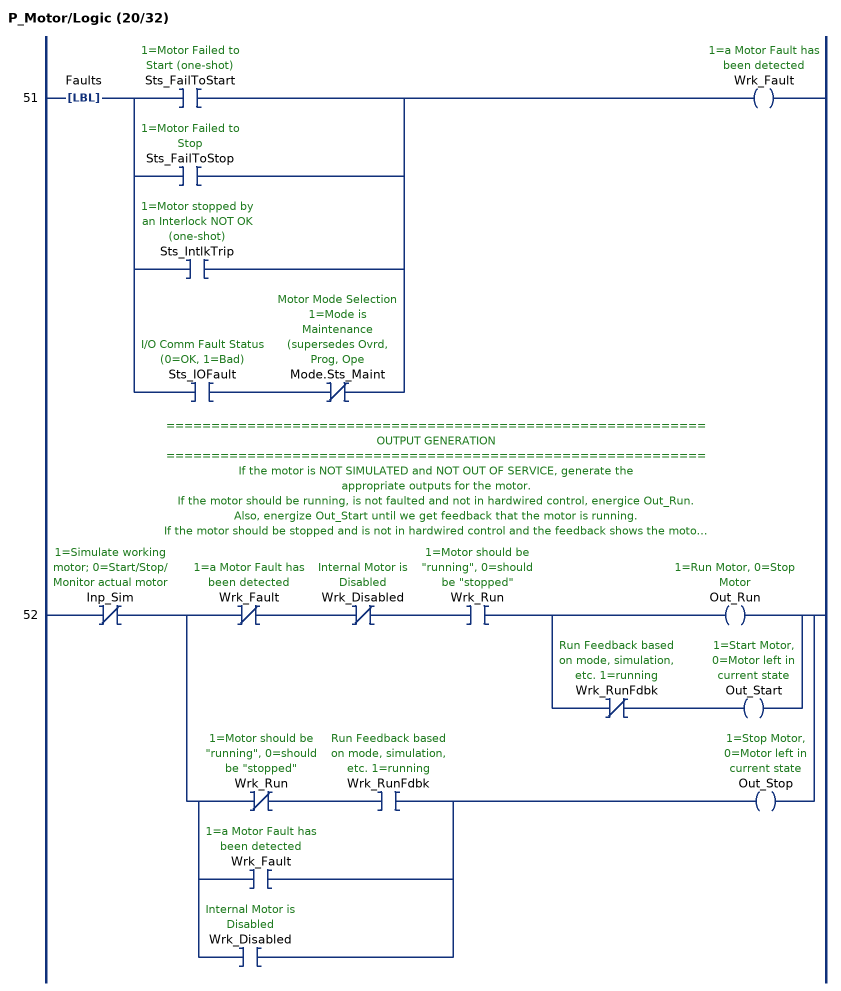
   51: LBL(Faults)[XIC(Sts_FailToStart) ,XIC(Sts_FailToStop) ,XIC(Sts_IntlkTrip) ,XIC(Sts_IOFault) XIO(Mode.Sts_Maint) ]OTE(Wrk_Fault);
   // ============================================================
   // OUTPUT GENERATION
   // ============================================================
   // If the motor is NOT SIMULATED and NOT OUT OF SERVICE, generate the
   // appropriate outputs for the motor.
   // If the motor should be running, is not faulted and not in hardwired control, energice Out_Run.
   // Also, energize Out_Start until we get feedback that the motor is running.
   // If the motor should be stopped and is not in hardwired control and the feedback shows the motor
   // is NOT stopped, or if the motor is Faulted, energize the Out_Stop output to stop the motor.
   52: XIO(Inp_Sim)[XIO(Wrk_Fault) XIO(Wrk_Disabled) XIC(Wrk_Run) [OTE(Out_Run) ,XIO(Wrk_RunFdbk) OTE(Out_Start) ] ,[XIO(Wrk_Run) XIC(Wrk_RunFdbk) ,XIC(Wrk_Fault) ,XIC(Wrk_Disabled) ] OTE(Out_Stop) ];
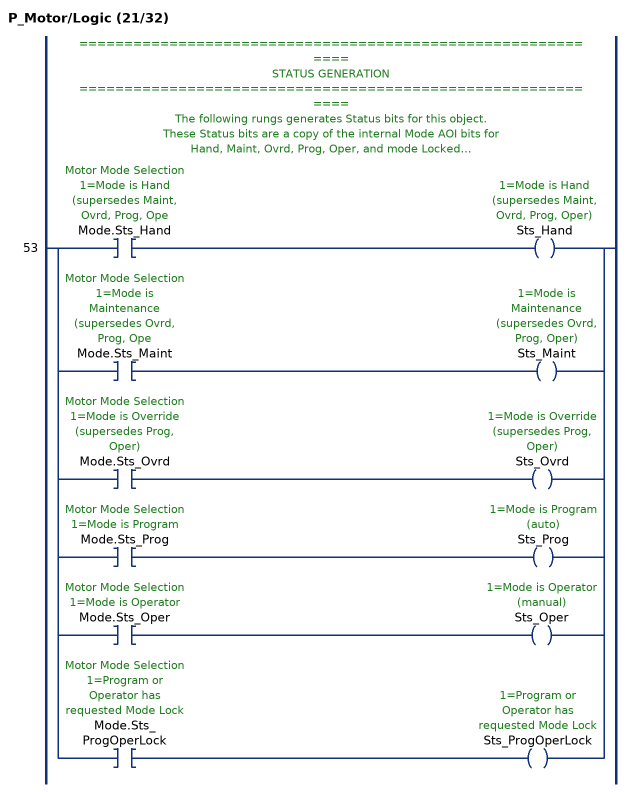
   // ============================================================
   // STATUS GENERATION
   // ============================================================
   // The following rungs generates Status bits for this object.
   // These Status bits are a copy of the internal Mode AOI bits for
   // Hand, Maint, Ovrd, Prog, Oper, and mode Locked.
   // NOTE for Sts_Maint:  This Motor is in Maintenance (Out Of Service, no able to run normally)
   // if this instruction is on a False Rung (Enable In False).  See the Enable In False Routine.
   53: [XIC(Mode.Sts_Hand) OTE(Sts_Hand) ,XIC(Mode.Sts_Maint) OTE(Sts_Maint) ,XIC(Mode.Sts_Ovrd) OTE(Sts_Ovrd) ,XIC(Mode.Sts_Prog) OTE(Sts_Prog) ,XIC(Mode.Sts_Oper) OTE(Sts_Oper) ,XIC(Mode.Sts_ProgOperLock) OTE(Sts_ProgOperLock) ];
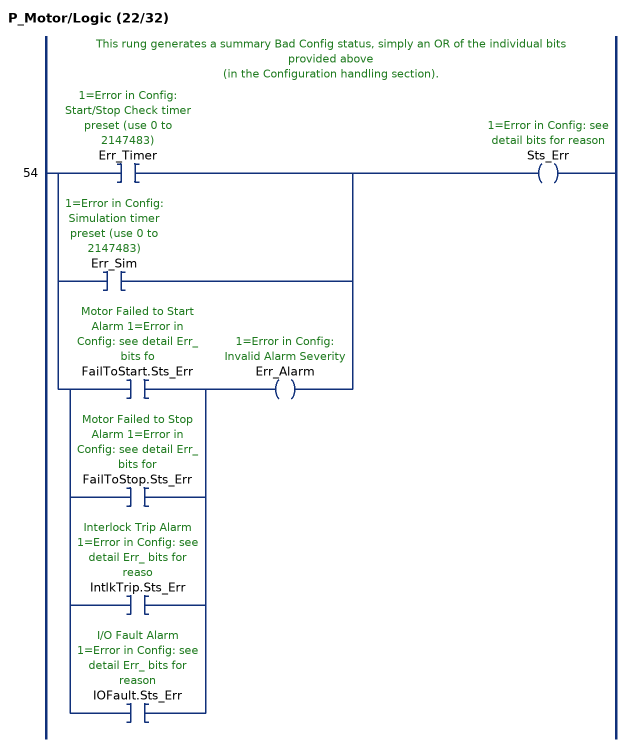
   // This rung generates a summary Bad Config status, simply an OR of the individual bits provided above
   // (in the Configuration handling section).
   54: [XIC(Err_Timer) ,XIC(Err_Sim) ,[XIC(FailToStart.Sts_Err) ,XIC(FailToStop.Sts_Err) ,XIC(IntlkTrip.Sts_Err) ,XIC(IOFault.Sts_Err) ] OTE(Err_Alarm) ]OTE(Sts_Err);
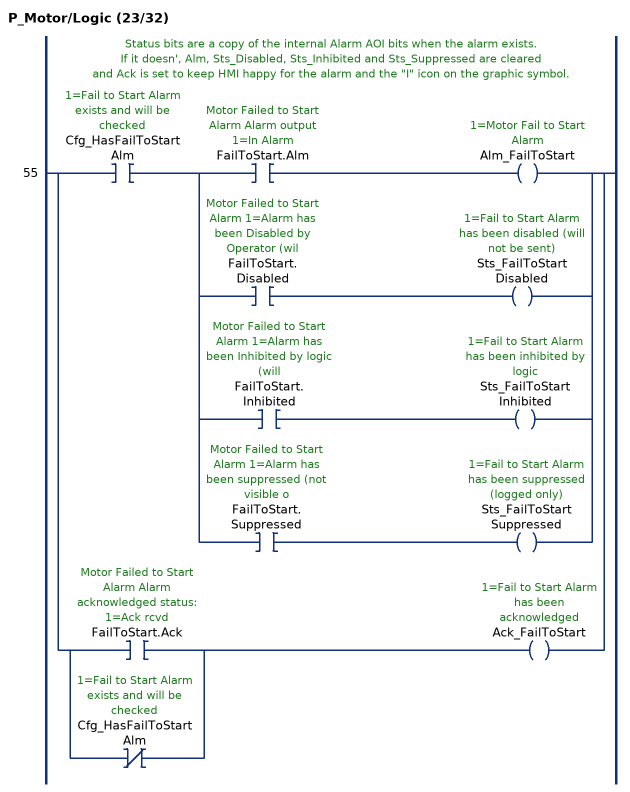
   // Status bits are a copy of the internal Alarm AOI bits when the alarm exists.
   // If it doesn', Alm, Sts_Disabled, Sts_Inhibited and Sts_Suppressed are cleared
   // and Ack is set to keep HMI happy for the alarm and the "I" icon on the graphic symbol.
   55: [XIC(Cfg_HasFailToStartAlm) [XIC(FailToStart.Alm) OTE(Alm_FailToStart) ,XIC(FailToStart.Disabled) OTE(Sts_FailToStartDisabled) ,XIC(FailToStart.Inhibited) OTE(Sts_FailToStartInhibited) ,XIC(FailToStart.Suppressed) OTE(Sts_FailToStartSuppressed) ] ,[XIC(FailToStart.Ack) ,XIO(Cfg_HasFailToStartAlm) ] OTE(Ack_FailToStart) ];
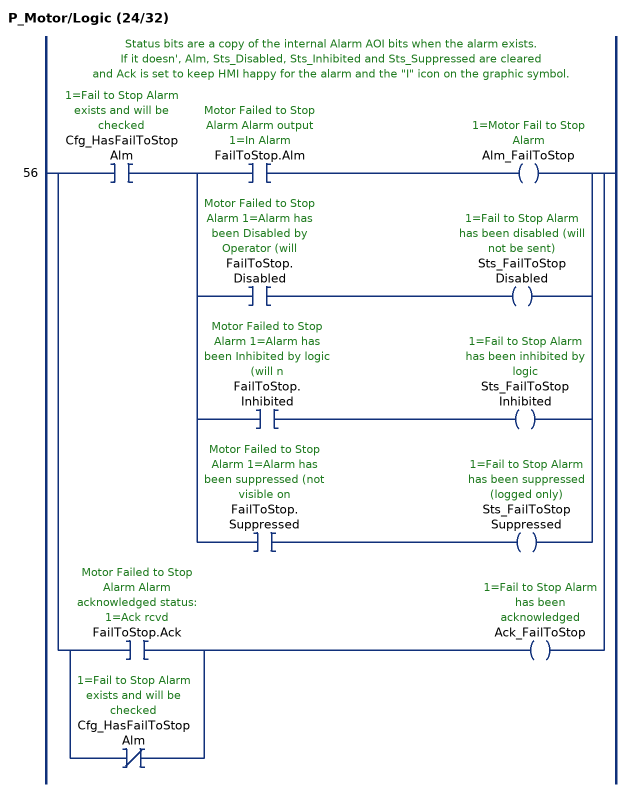
   // Status bits are a copy of the internal Alarm AOI bits when the alarm exists.
   // If it doesn', Alm, Sts_Disabled, Sts_Inhibited and Sts_Suppressed are cleared
   // and Ack is set to keep HMI happy for the alarm and the "I" icon on the graphic symbol.
   56: [XIC(Cfg_HasFailToStopAlm) [XIC(FailToStop.Alm) OTE(Alm_FailToStop) ,XIC(FailToStop.Disabled) OTE(Sts_FailToStopDisabled) ,XIC(FailToStop.Inhibited) OTE(Sts_FailToStopInhibited) ,XIC(FailToStop.Suppressed) OTE(Sts_FailToStopSuppressed) ] ,[XIC(FailToStop.Ack) ,XIO(Cfg_HasFailToStopAlm) ] OTE(Ack_FailToStop) ];
